TYPE csp_case_loader_rfid_status_enum :
(
	CSP_CASE_LOADER_RFID_STATUS_START 							:= 1,
	CSP_CASE_LOADER_RFID_STATUS_CHECK_AXIS_POS					:= 5,
	CSP_CASE_LOADER_RFID_STATUS_DISABLE_AXIS					:= 10,
	CSP_CASE_LOADER_RFID_STATUS_ENABLE_AXIS						:= 20,
	CSP_CASE_LOADER_RFID_STATUS_ENABLE_CROSSPUSHERS				:= 21,
	CSP_CASE_LOADER_RFID_STATUS_MOVE_CROSSPUSHERS				:= 22,
	CSP_CASE_LOADER_RFID_VERIFY_CROSSPUSHERS_CLEAR				:= 25,
	CSP_CASE_LOADER_RFID_STATUS_MOVE_AXIS_TO_POS				:= 30,
	CSP_CASE_LOADER_RFID_STATUS_VERIFY_AXIS_POS					:= 40,
	
	CSP_CASE_LOADER_RFID_STATUS_CHECK_READ_WRITE				:= 50,
	
	CSP_CASE_LOADER_RFID_STATUS_READ_START						:= 100,
	CSP_CASE_LOADER_RFID_STATUS_READ_CHECK_RESULT				:= 110,
	CSP_CASE_LOADER_RFID_STATUS_READ_DONE						:= 120,
	
	CSP_CASE_LOADER_RFID_STATUS_WRITE_START						:= 200,
	CSP_CASE_LOADER_RFID_STATUS_WAIT_WRITE						:= 210,
	CSP_CASE_LOADER_RFID_STATUS_WRITE_DONE						:= 220,
	
	
	CSP_CASE_LOADER_RFID_STATUS_WAITING							:= 900
) := CSP_CASE_LOADER_RFID_STATUS_WAITING;
END_TYPE

(* stored: Version 1.1.0.1, ProductVersion 3.1.4024.3
   DUT csp_case_loader_rfid_status_enum: Id {0c3dbfa2-39b5-47fd-850f-2cdd70310f0a} *)
